// TwinCAT 3 PLC project CSVExample
// ProgramVersion: 3.1.0.8
// libraries:
//   Tc2_Standard, * (Beckhoff Automation GmbH)
//   Tc2_System, * (Beckhoff Automation GmbH)
//   Tc2_Utilities, * (Beckhoff Automation GmbH)
//   Tc3_Interfaces, * (Beckhoff Automation GmbH)
//   Tc3_Module, * (Beckhoff Automation GmbH)
// project tree:
//   DUTs/ ST_CSV_Record.TcDUT (not stored)
//   GVLs/ GVL.TcGVL (not stored), GVL_1.TcGVL, GVL_2.TcGVL
//   POUs/CSV read_write in binary mode/ P_BinaryModeRead.TcPOU (not stored), P_BinaryModeWrite.TcPOU (not stored)
//   POUs/CSV read_write in text mode/ P_TextModeRead.TcPOU (not stored), P_TextModeWrite.TcPOU (not stored)
//   POUs/ MAIN.TcPOU (not stored), P_ArgToConvExample.TcPOU (not stored), P_StringToConvExample.TcPOU (not stored)
//   / PlcTask.TcTTO (not stored)
// real-time tasks:
//   TASK PlcTask: cycle T#10ms, priority 20, ADS port 350
//   TASK PlcTask1: cycle T#10ms, priority 21, ADS port 351

// ---- GVLs/GVL_1.TcGVL
{attribute 'qualified_only'}
VAR_GLOBAL
END_VAR

// ---- GVLs/GVL_2.TcGVL
{attribute 'qualified_only'}
VAR_GLOBAL
END_VAR
